FUNCTION_BLOCK PUBLIC FB_TrafficLightController
VAR
	nNumberOfTrafficLights : SINT;
	currentLight: SINT := 1;
	
	arTrafficLights: ARRAY[1..4] OF FB_TrafficLight;
	arTrafficLightsInvisible: ARRAY[1..4] OF BOOL;
	
END_VAR

StartCurrentTrafficLight();

RefereshAllTrafficLights();

TrySwitchToNextTrafficLight();

PROPERTY PUBLIC NumberOfTrafficLights : SINT
GET
NumberOfTrafficLights := nNumberOfTrafficLights;
END_GET
SET
IF NumberOfTrafficLights >= 2 AND NumberOfTrafficLights <= 4 THEN
	nNumberOfTrafficLights := NumberOfTrafficLights;
	SetVisibleTrafficLights();
END_IF
END_SET
END_PROPERTY

METHOD PRIVATE RefereshAllTrafficLights
VAR
	index: SINT;
END_VAR
FOR index := 1 TO nNumberOfTrafficLights DO
	arTrafficLights[index]();
END_FOR
END_METHOD

METHOD PUBLIC Setup
VAR_INPUT
	lightNumber: SINT;
	
	redDuration: TIME;
	yellowDuration: TIME;
	greenDuration: TIME;
END_VAR
IF lightNumber >= 1 AND lightNumber <= GVL.MAX_TRAFFIC_LIGHTS THEN
	arTrafficLights[lightNumber].Setup(redDuration, yellowDuration, greenDuration);
END_IF
END_METHOD

METHOD PRIVATE SetVisibleTrafficLights
VAR
	idx: INT;
END_VAR
FOR idx := 1 TO GVL.MAX_TRAFFIC_LIGHTS DO
	arTrafficLightsInvisible[idx] := TRUE;
END_FOR

FOR idx := 1 TO nNumberOfTrafficLights DO
	arTrafficLightsInvisible[idx] := FALSE;
END_FOR
END_METHOD

METHOD PRIVATE StartCurrentTrafficLight
IF NOT arTrafficLights[currentLight].Start THEN
	arTrafficLights[currentLight].Start := TRUE;
END_IF
END_METHOD

METHOD PRIVATE TrySwitchToNextTrafficLight
IF arTrafficLights[currentLight].CanSwitch() THEN
	currentLight := currentLight + 1;
	IF currentLight > nNumberOfTrafficLights THEN
		currentLight := 1;
	END_IF
END_IF
END_METHOD

END_FUNCTION_BLOCK

(* stored: Version 1.1.0.1, ProductVersion 3.1.4024.12
   POU FB_TrafficLightController: Id {3fc0ac03-c5fc-49e7-9c92-f062a7fda4fa}, SpecialFunc None
   Property NumberOfTrafficLights: Id {687c6475-ec52-440a-b0b5-00ed78dcc3ef}
   Get Get: Id {ad8de530-6fc0-4c75-ada0-fed0b8927409}
   Set Set: Id {2bcee6ce-e8dd-40bd-9a16-8f25ee7518b9}
   Method RefereshAllTrafficLights: Id {2288413a-7e69-49e8-a317-93a1c9b50390}
   Method Setup: Id {24b403de-5e34-452f-a034-12bcc6c30339}
   Method SetVisibleTrafficLights: Id {4e8082c2-1ae0-484b-a686-00360c7b93e5}
   Method StartCurrentTrafficLight: Id {64998691-cd67-45c5-8343-719572b9dc57}
   Method TrySwitchToNextTrafficLight: Id {904086e1-c5fb-441f-adf7-b574b1cbcdc5} *)
